INTERFACE ITF_BaseLogger_HMI_Connector EXTENDS ITF_BaseLogger_HMI_Connector_Command, ITF_BaseLogger_HMI_Connector_View

END_INTERFACE

(* stored: Version 1.1.0.1
   Itf ITF_BaseLogger_HMI_Connector: Id {95c86d1b-cfc8-07b1-10e7-5e8303503e4e} *)
